// TIA Portal V17 export
// export: Created 2022-07-20T06:59:50.2887268Z, ExportSetting WithDefaults, DisplayName Totally Integrated Automation Portal, DisplayVersion V17, DisplayName TIA Portal Openness, DisplayVersion V17, DisplayName TIA Portal Version Control Interface, DisplayVersion V17, DisplayName SINAMICS Startdrive Advanced, DisplayVersion V17, DisplayName SINAMICS Startdrive G130, G150, S120, S150, SINAMICS MV, S210, DisplayVersion V17, DisplayName SINAMICS Startdrive G110M, G120, G120C, G120D, G120P, G115D, DisplayVersion V17, DisplayName STEP 7 Professional, DisplayVersion V17, DisplayName STEP 7 Safety, DisplayVersion V17, DisplayName WinCC Advanced, DisplayVersion V17
FUNCTION_BLOCK "FB10060_IperPrintingInkCircuit"   // FB10060, LAD
{ S7_Optimized_Access := 'TRUE' }
VERSION : 0.1
// Hauteur du Tank 115mm
// Zone du capteur 97mm
// stored: AutoNumber false, IsIECCheckEnabled false, IsRetainMemResEnabled false, MemoryReserve 100, SetENOAutomatically false, UDAEnableTagReadback false
   VAR_INPUT
      Sensor_Value : Int;
      Sensor_HighErrorThreshold : Real;
      Sensor_HighWarningThreshold : Real;
      Sensor_LowWarningThreshold : Real;
      Sensor_LowErrorThreshold : Real;
      BarrelWS_RawValue : Int;
      BarrelWS_CalibrationValue_1 : Real;
      BarrelWS_CalibrationValue_2 : Real;
      BarrelWS_LowWarningThreshold : Real;
      BarrelWS_HighWarningThreshold : Real;
      BarrelWS_LowErrorThreshold : Real;
      BarrelWS_HighErrorThreshold : Real;
      Tank_ReachLevel : Real;
      Tank_RegulationLevel : Real;
      SystemPressurized : Bool;
      SystemDepressurized : Bool;
   END_VAR
   VAR_OUTPUT
      ActivePump : Bool;
      PumpDirection : Bool;
      ActiveGeneralSolenoid : Bool;
      ActiveFillingSolenoid : Bool;
      BarrelWS_CalibrationStatus_1 : Bool;
      BarrelWS_CalibrationStatus_2 : Bool;
      BarrelWS_LowWarningThresholdReached : Bool;
      BarrelWS_HighWarningThresholdReached : Bool;
      BarrelWS_LowErrorThresholdReached : Bool;
      BarrelWS_HighErrorThresholdReached : Bool;
      BarrelWS_NetWeight : Real;
      "BarrelWS_NetWeight_%" : Real;
      BarrelWS_CalibrationDone : Bool;
      Tank_VarnishQuantity_mm : Real;
      "Tank_VarnishQuantity_%" : Real;
      Tank_ReachLevelDone : Bool;
      Tank_AutoRegulationInProgress : Bool;
      Sensor_HighErrorThresholdReached : Bool;
      Sensor_HighWarningThresholdReached : Bool;
      Sensor_LowWarningThresholdReached : Bool;
      Sensor_LowErrorThresholdReached : Bool;
      Sensor_Calibrated : Bool;
      InkCircuitInError : Bool;
      AutoRegulationPositionDeviationDetected : Bool;
   END_VAR
   VAR_IN_OUT
      RequestAcknowledge : Bool;
      BarrelWS_RequestCalibration_1 : Bool;
      BarrelWS_RequestCalibration_2 : Bool;
      Tank_RequestReachLevel : Bool;
      Tank_RequestActiveAutoRegulation : Bool;
      BarrelWS_ResetCalibration : Bool;
      Sensor_CalibrationValueX_1 : Real;
      Sensor_CalibrationValueY_1 : Real;
      Sensor_CalibrationValueX_2 : Real;
      Sensor_CalibrationValueY_2 : Real;
      BarrelWS_CalibrationDataX_1 : Real;
      BarrelWS_CalibrationDataY_1 : Real;
      BarrelWS_CalibrationDataX_2 : Real;
      BarrelWS_CalibrationDataY_2 : Real;
   END_VAR
   VAR
      DirectionSended : Bool;
      AutoRegulationReachedLevelOnce : Bool;
      InkTankOperationStateDiagram : Int;
      R_TRIG_FillTank : R_TRIG;
      R_TRIG_DrainTank { S7_SetPoint := 'True'} : R_TRIG;
      R_TRIG_ReachLevelTank { S7_SetPoint := 'True'} : R_TRIG;
      R_TRIG_AutoRegulation { S7_SetPoint := 'True'} : R_TRIG;
      F_TRIG_FillTank { S7_SetPoint := 'True'} : F_TRIG;
      F_TRIG_DrainTank { S7_SetPoint := 'True'} : F_TRIG;
      F_TRIG_ReachLevelTank { S7_SetPoint := 'True'} : F_TRIG;
      F_TRIG_AutoRegulation { S7_SetPoint := 'True'} : F_TRIG;
      TON_AutoRegulationPositionDeviation { S7_SetPoint := 'True'} : TON_TIME;
      TON_SendActivationAfterDirection { S7_SetPoint := 'True'} : TON_TIME;
      TON_FillTankSafety { S7_SetPoint := 'True'} : TON_TIME;
      TON_OverPressure { S7_SetPoint := 'True'} : TON_TIME;
      FB10030_AnalogicalSensor_MicrosonicUltrasonicSensor_TankLevel { S7_SetPoint := 'True'} : "FB10030_AnalogicalSensor";
      FB10030_AnalogicalSensor_TLMScale_VarnishBarrel { S7_SetPoint := 'True'} : "FB10030_AnalogicalSensor";
   END_VAR
   VAR CONSTANT
      WAIT_FOR_OPERATION_REQUEST : Int := 0;
      FILL_TANK : Int := 10;
      DRAIN_TANK : Int := 20;
      REACH_LEVEL_TANK : Int := 30;
      AUTO_REGULATION : Int := 40;
      OPERATION_DONE : Int := 50;
   END_VAR
BEGIN

REGION Network 1 (SCL): First Scan
   IF "FirstScan" THEN
       #DirectionSended := FALSE;
       #Tank_ReachLevelDone := FALSE;
       #InkTankOperationStateDiagram := #WAIT_FOR_OPERATION_REQUEST;
   END_IF;
END_REGION

REGION Network 2 (SCL): Edge Signals & Timers
   REGION EDGE SIGNALS
       #R_TRIG_ReachLevelTank(CLK := #Tank_RequestReachLevel);
       #R_TRIG_AutoRegulation(CLK := #Tank_RequestActiveAutoRegulation);

       #F_TRIG_ReachLevelTank(CLK := #Tank_RequestReachLevel);
       #F_TRIG_AutoRegulation(CLK := #Tank_RequestActiveAutoRegulation);
   END_REGION

   REGION TIMERS
       #TON_AutoRegulationPositionDeviation(IN := #AutoRegulationReachedLevelOnce AND NOT ("FC10021_TolerenceRelation"(X := #Tank_VarnishQuantity_mm, Y := #Tank_RegulationLevel, Tolerance := 10.0)),
                                            PT := T#5s);
       #TON_SendActivationAfterDirection(IN := #InkTankOperationStateDiagram = #FILL_TANK OR
                                         #InkTankOperationStateDiagram = #DRAIN_TANK OR
                                         #InkTankOperationStateDiagram = #REACH_LEVEL_TANK OR
                                         #InkTankOperationStateDiagram = #AUTO_REGULATION,
                                         PT := T#20ms); //Time direction signal sended and pump activation necessary for the electronical card
       #TON_FillTankSafety(IN := #ActivePump AND #PumpDirection,
                           PT := T#380s);  
   END_REGION
END_REGION

REGION Network 3 (SCL): Tank Commands Management
   IF #TON_SendActivationAfterDirection.Q THEN
       #DirectionSended := TRUE;
   END_IF;
END_REGION

REGION Network 4: Ink Barrel Weigh Scale Management
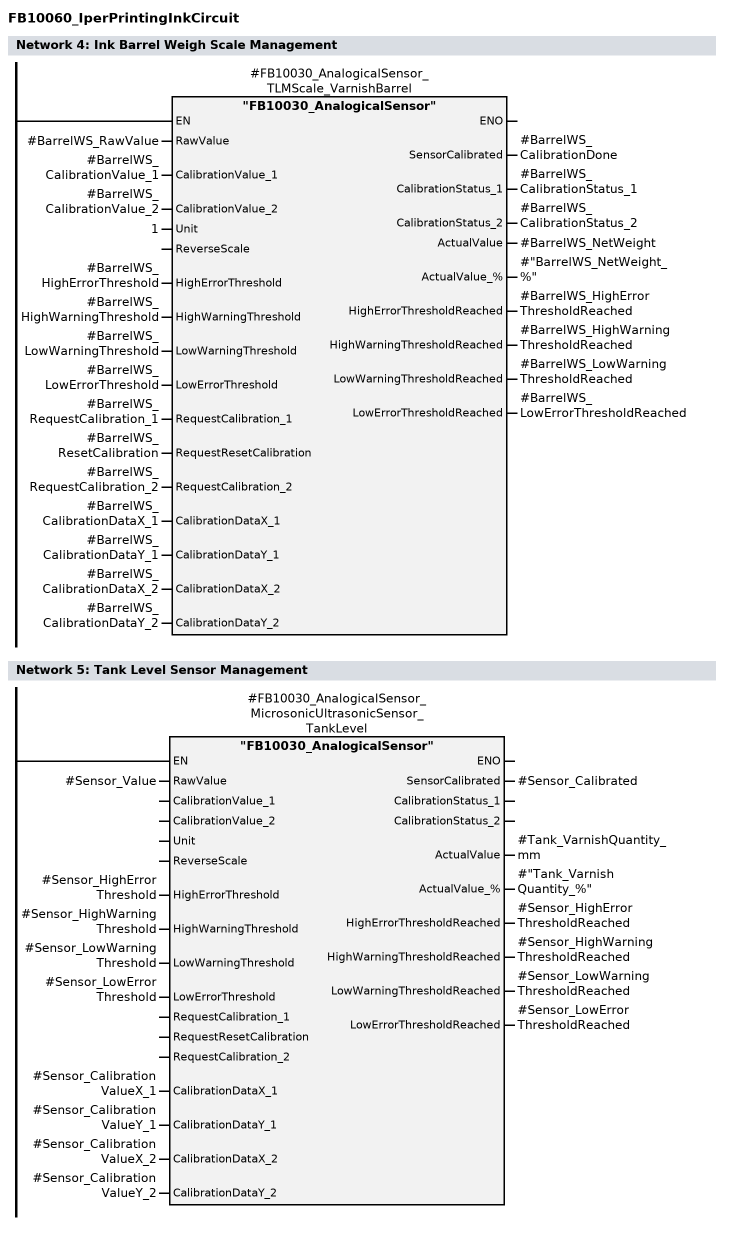
   RUNG wire#powerrail
      #FB10030_AnalogicalSensor_TLMScale_VarnishBarrel(RawValue := #BarrelWS_RawValue, CalibrationValue_1 := #BarrelWS_CalibrationValue_1, CalibrationValue_2 := #BarrelWS_CalibrationValue_2, Unit := 1, ReverseScale :=, HighErrorThreshold := #BarrelWS_HighErrorThreshold, HighWarningThreshold := #BarrelWS_HighWarningThreshold, LowWarningThreshold := #BarrelWS_LowWarningThreshold, LowErrorThreshold := #BarrelWS_LowErrorThreshold, RequestCalibration_1 := #BarrelWS_RequestCalibration_1, RequestCalibration_2 := #BarrelWS_RequestCalibration_2, RequestResetCalibration := #BarrelWS_ResetCalibration, CalibrationDataX_1 := #BarrelWS_CalibrationDataX_1, CalibrationDataY_1 := #BarrelWS_CalibrationDataY_1, CalibrationDataX_2 := #BarrelWS_CalibrationDataX_2, CalibrationDataY_2 := #BarrelWS_CalibrationDataY_2, SensorCalibrated => #BarrelWS_CalibrationDone, CalibrationStatus_1 => #BarrelWS_CalibrationStatus_1, CalibrationStatus_2 => #BarrelWS_CalibrationStatus_2, ActualValue => #BarrelWS_NetWeight, "ActualValue_%" => #"BarrelWS_NetWeight_%", HighErrorThresholdReached => #BarrelWS_HighErrorThresholdReached, HighWarningThresholdReached => #BarrelWS_HighWarningThresholdReached, LowWarningThresholdReached => #BarrelWS_LowWarningThresholdReached, LowErrorThresholdReached => #BarrelWS_LowErrorThresholdReached)
   END_RUNG
   // the same network as SCL:
   #FB10030_AnalogicalSensor_TLMScale_VarnishBarrel(RawValue := #BarrelWS_RawValue,   // "FB10030_AnalogicalSensor"
                           CalibrationValue_1 := #BarrelWS_CalibrationValue_1,
                           CalibrationValue_2 := #BarrelWS_CalibrationValue_2,
                           Unit := 1,
                           HighErrorThreshold := #BarrelWS_HighErrorThreshold,
                           HighWarningThreshold := #BarrelWS_HighWarningThreshold,
                           LowWarningThreshold := #BarrelWS_LowWarningThreshold,
                           LowErrorThreshold := #BarrelWS_LowErrorThreshold,
                           RequestCalibration_1 := #BarrelWS_RequestCalibration_1,
                           RequestResetCalibration := #BarrelWS_ResetCalibration,
                           RequestCalibration_2 := #BarrelWS_RequestCalibration_2,
                           CalibrationDataX_1 := #BarrelWS_CalibrationDataX_1,
                           CalibrationDataY_1 := #BarrelWS_CalibrationDataY_1,
                           CalibrationDataX_2 := #BarrelWS_CalibrationDataX_2,
                           CalibrationDataY_2 := #BarrelWS_CalibrationDataY_2,
                           SensorCalibrated => #BarrelWS_CalibrationDone,
                           CalibrationStatus_1 => #BarrelWS_CalibrationStatus_1,
                           CalibrationStatus_2 => #BarrelWS_CalibrationStatus_2,
                           ActualValue => #BarrelWS_NetWeight,
                           "ActualValue_%" => #"BarrelWS_NetWeight_%",
                           HighErrorThresholdReached => #BarrelWS_HighErrorThresholdReached,
                           HighWarningThresholdReached => #BarrelWS_HighWarningThresholdReached,
                           LowWarningThresholdReached => #BarrelWS_LowWarningThresholdReached,
                           LowErrorThresholdReached => #BarrelWS_LowErrorThresholdReached);
END_REGION

REGION Network 5: Tank Level Sensor Management
   RUNG wire#powerrail
      #FB10030_AnalogicalSensor_MicrosonicUltrasonicSensor_TankLevel(RawValue := #Sensor_Value, CalibrationValue_1 :=, CalibrationValue_2 :=, Unit :=, ReverseScale :=, HighErrorThreshold := #Sensor_HighErrorThreshold, HighWarningThreshold := #Sensor_HighWarningThreshold, LowWarningThreshold := #Sensor_LowWarningThreshold, LowErrorThreshold := #Sensor_LowErrorThreshold, RequestCalibration_1 :=, RequestCalibration_2 :=, RequestResetCalibration :=, CalibrationDataX_1 := #Sensor_CalibrationValueX_1, CalibrationDataY_1 := #Sensor_CalibrationValueY_1, CalibrationDataX_2 := #Sensor_CalibrationValueX_2, CalibrationDataY_2 := #Sensor_CalibrationValueY_2, SensorCalibrated => #Sensor_Calibrated, CalibrationStatus_1 =>, CalibrationStatus_2 =>, ActualValue => #Tank_VarnishQuantity_mm, "ActualValue_%" => #"Tank_VarnishQuantity_%", HighErrorThresholdReached => #Sensor_HighErrorThresholdReached, HighWarningThresholdReached => #Sensor_HighWarningThresholdReached, LowWarningThresholdReached => #Sensor_LowWarningThresholdReached, LowErrorThresholdReached => #Sensor_LowErrorThresholdReached)
   END_RUNG
   // the same network as SCL:
   #FB10030_AnalogicalSensor_MicrosonicUltrasonicSensor_TankLevel(RawValue := #Sensor_Value,   // "FB10030_AnalogicalSensor"
                           HighErrorThreshold := #Sensor_HighErrorThreshold,
                           HighWarningThreshold := #Sensor_HighWarningThreshold,
                           LowWarningThreshold := #Sensor_LowWarningThreshold,
                           LowErrorThreshold := #Sensor_LowErrorThreshold,
                           CalibrationDataX_1 := #Sensor_CalibrationValueX_1,
                           CalibrationDataY_1 := #Sensor_CalibrationValueY_1,
                           CalibrationDataX_2 := #Sensor_CalibrationValueX_2,
                           CalibrationDataY_2 := #Sensor_CalibrationValueY_2,
                           SensorCalibrated => #Sensor_Calibrated,
                           ActualValue => #Tank_VarnishQuantity_mm,
                           "ActualValue_%" => #"Tank_VarnishQuantity_%",
                           HighErrorThresholdReached => #Sensor_HighErrorThresholdReached,
                           HighWarningThresholdReached => #Sensor_HighWarningThresholdReached,
                           LowWarningThresholdReached => #Sensor_LowWarningThresholdReached,
                           LowErrorThresholdReached => #Sensor_LowErrorThresholdReached);
END_REGION

REGION Network 6 (SCL): Tank Ink Management
   CASE #InkTankOperationStateDiagram OF
       #WAIT_FOR_OPERATION_REQUEST:
           IF #R_TRIG_ReachLevelTank.Q THEN
               #Tank_ReachLevelDone := FALSE;
               #PumpDirection := TRUE;
               #InkTankOperationStateDiagram := #REACH_LEVEL_TANK;
           ELSIF #R_TRIG_AutoRegulation.Q THEN
               #Tank_ReachLevelDone := FALSE;
               #PumpDirection := FALSE;
               #InkTankOperationStateDiagram := #AUTO_REGULATION;
           END_IF;
       #REACH_LEVEL_TANK:
           //Signals Management
           IF #DirectionSended THEN
               #ActivePump := TRUE;
               IF #Tank_VarnishQuantity_mm >= #Tank_ReachLevel THEN
                   #ActiveGeneralSolenoid := TRUE;
                   #ActiveFillingSolenoid := TRUE;
                   #PumpDirection := FALSE;
               ELSIF #Tank_VarnishQuantity_mm < #Tank_ReachLevel THEN
                   #ActiveGeneralSolenoid := FALSE;
                   #ActiveFillingSolenoid := TRUE;
                   #PumpDirection := TRUE;
               END_IF;
           END_IF;

           //Condition To Go To Next Step
           IF
               "FC10021_TolerenceRelation"(X := #Tank_VarnishQuantity_mm, Y := #Tank_ReachLevel, Tolerance := 0.1) OR
               #F_TRIG_ReachLevelTank.Q
           THEN
               #ActiveGeneralSolenoid := FALSE;
               #ActiveFillingSolenoid := FALSE;
               #ActivePump := FALSE;
               #PumpDirection := FALSE;
               #Tank_ReachLevelDone := TRUE;
               #DirectionSended := FALSE;
               RESET_TIMER(#TON_SendActivationAfterDirection);
               #InkTankOperationStateDiagram := #OPERATION_DONE;
           END_IF;
       #AUTO_REGULATION:
           //Signals Management
           #Tank_AutoRegulationInProgress := TRUE;
           IF #DirectionSended THEN
               IF #Tank_VarnishQuantity_mm >= #Tank_RegulationLevel THEN
                   #ActivePump := FALSE;
                   #ActiveGeneralSolenoid := FALSE;
                   #ActiveFillingSolenoid := FALSE;
                   #AutoRegulationReachedLevelOnce := TRUE;
               ELSIF #Tank_VarnishQuantity_mm < #Tank_RegulationLevel - 1.0 THEN
                   #ActivePump := TRUE;
                   #ActiveGeneralSolenoid := FALSE;
                   #ActiveFillingSolenoid := TRUE;
                   #PumpDirection := TRUE;
                   #AutoRegulationReachedLevelOnce := FALSE;
               END_IF;
           END_IF;

           //Condition To Go to Next Step
           IF #F_TRIG_AutoRegulation.Q OR #TON_FillTankSafety.Q THEN
               #Tank_AutoRegulationInProgress := FALSE;
               #ActiveGeneralSolenoid := FALSE;
               #ActiveFillingSolenoid := FALSE;
               #ActivePump := FALSE;
               #PumpDirection := FALSE;
               #DirectionSended := FALSE;
               #AutoRegulationReachedLevelOnce := FALSE;
               RESET_TIMER(#TON_SendActivationAfterDirection);
               #InkTankOperationStateDiagram := #OPERATION_DONE;
           END_IF;
       #OPERATION_DONE:
           #InkTankOperationStateDiagram := #WAIT_FOR_OPERATION_REQUEST;
   END_CASE;
END_REGION

REGION Network 7 (SCL): Error Management
   //Ink Circuit Error Management
   IF #TON_FillTankSafety.Q OR #Sensor_Value < 200.0 OR NOT(#Sensor_Calibrated) OR NOT(#BarrelWS_CalibrationDone) THEN
       #InkCircuitInError := TRUE;
   ELSIF #RequestAcknowledge THEN
       #InkCircuitInError := FALSE;
   END_IF;

   //Auto Regulation Position Deviation Error Management
   IF #TON_AutoRegulationPositionDeviation.Q THEN
       #AutoRegulationPositionDeviationDetected := TRUE;
   ELSIF #RequestAcknowledge THEN
       #AutoRegulationPositionDeviationDetected := FALSE;
   END_IF;
END_REGION
END_FUNCTION_BLOCK
